TEXTLIST nPlcEventID
  0 = ''
  1 = 'Alarm Mesaji - 1' | English: 'Alarm Message - 1' | Turkish: 'Alarm Mesaji - 1'
  2 = 'Uyari Mesaji - 1' | English: 'Warning Message -1' | Turkish: 'Uyari Mesaji - 1'
  3 = 'Sicaklik Hatasi-2' | English: 'Temp Error-1' | Turkish: 'Sicaklik Hatasi-1'
  4 = 'BASINC HATASI' | English: 'PRESSURE ERROR' | Turkish: 'BASINC HATASI'
   = ''
END_TEXTLIST

(* stored: Version 1.1.0.1, ProductVersion 3.1.4024.6
   TextList nPlcEventID: Id {ebeb7edf-c613-4367-9ae9-967bfbe1b60e} *)
